(* Logix 5000 project; controller EuniceF_ICA5 vendor 1 type 14 code 150 rev 37.11; software revision 37.00 *)

TASK MainTask (continuous, watchdog 500 ms) : MainProgram

MODULES
   Local : vendor 1 type 14 code 150 (Compact 0, rev 37.11)
      Discrete_IO : Embedded (Compact 1, rev 3.1, Output RPI 20 ms)
      Analog_IO : Embedded (Compact 2, rev 1.1, Output RPI 80 ms)
      Counters : Embedded (Compact 3, rev 1.1, Output RPI 20 ms)
END_MODULES

VAR_GLOBAL   (* controller tags *)
   COIL1 : BOOL;
   COIL2 : BOOL;
   START : BOOL;
   STOP : BOOL;
END_VAR

PROGRAM MainProgram   (* main routine MainRoutine *)

ROUTINE MainRoutine   (* ladder *)
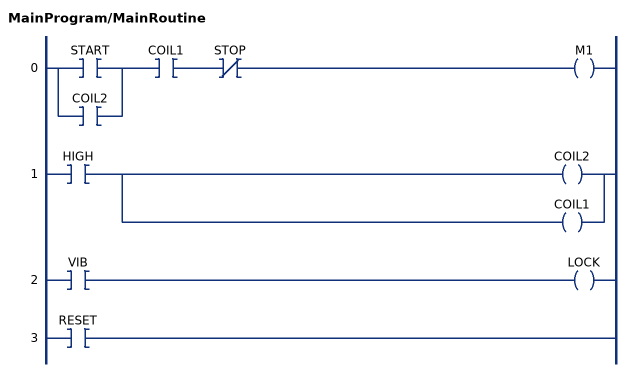
   0: [XIC(START) ,XIC(COIL2) ]XIC(COIL1)XIO(STOP)OTE(M1);
   1: XIC(HIGH)[OTE(COIL2) ,OTE(COIL1) ];
   2: XIC(VIB)OTE(LOCK);
   3: XIC(RESET);
END_ROUTINE
END_PROGRAM
